PROGRAM READ_VEL
VAR
	MC_ReadActualVelocity1 : MC_ReadActualVelocity;
	MC_ReadActualVelocity2 : MC_ReadActualVelocity;
	MC_ReadActualVelocity3 : MC_ReadActualVelocity;
	MC_ReadActualVelocity4 : MC_ReadActualVelocity;
END_VAR

MC_ReadActualVelocity1(
	Axis:= AXIS.Axis1, 
	Enable:= , 
	Valid=> , 
	Busy=> , 
	Error=> , 
	ErrorID=> , 
	ActualVelocity=> );
	
MC_ReadActualVelocity2(
	Axis:= AXIS.Axis2, 
	Enable:= , 
	Valid=> , 
	Busy=> , 
	Error=> , 
	ErrorID=> , 
	ActualVelocity=> );
	
MC_ReadActualVelocity3(
	Axis:= AXIS.Axis3, 
	Enable:= , 
	Valid=> , 
	Busy=> , 
	Error=> , 
	ErrorID=> , 
	ActualVelocity=> );
	
MC_ReadActualVelocity4(
	Axis:= AXIS.Axis4, 
	Enable:= , 
	Valid=> , 
	Busy=> , 
	Error=> , 
	ErrorID=> , 
	ActualVelocity=> );

END_PROGRAM

(* stored: Version 1.1.0.1, ProductVersion 3.1.4024.0
   POU READ_VEL: Id {1d381ed3-d54a-42ea-9667-e72b6bee0617}, SpecialFunc None *)
